{attribute 'GeneratedUsingTerminal: EL5002-0000-0016'}
{attribute addProperty BoxType "EL5002-0000-0016"}
{attribute addProperty Id "SSI_Inputs_Channel_1AT %I*SSI_Inputs_Channel_0E3D8E3310SSI_Inputs_Channel_2AT %I*SSI_Inputs_Channel_0E3D8E3310WcStateAT %I*WcState_9091E0EB2InfoDataAT %I*InfoData_94A18F5E2"}
{attribute addProperty CRC "177564199"}
{attribute addProperty Size "24"}
TYPE EL5002_0A956A27 EXTENDS EtcSlaveTerminalBase_947E5A46 :
STRUCT
	{attribute addProperty Name "SSI_Inputs_Channel_1"}
	SSI_Inputs_Channel_1 : SSI_Inputs_Channel_0E3D8E33;
	{attribute addProperty Name "SSI_Inputs_Channel_2"}
	SSI_Inputs_Channel_2 : SSI_Inputs_Channel_0E3D8E33;
	{attribute addProperty Name "WcState"}
	WcState : WcState_9091E0EB;
	{attribute addProperty Name "InfoData"}
	InfoData : InfoData_94A18F5E;
END_STRUCT
END_TYPE

(* stored: Version 1.2.0.0, ProductVersion 3.1.4024.9
   DUT EL5002_0A956A27: Id {330996fa-2596-4eb5-a80d-a74b13651c50} *)
